FUNCTION_BLOCK FB_EventIoTExporter IMPLEMENTS InterfaceEventViewer
VAR_INPUT
	tzinfo : ST_TimeZoneInformation;
END_VAR
VAR_OUTPUT
	export_event : ST_EventView;
END_VAR
VAR
END_VAR

{warning 'add method implementation '}
METHOD clear : BOOL
END_METHOD

{warning 'add method implementation '}
METHOD history_clear : BOOL
END_METHOD

{warning 'add method implementation '}
METHOD send_event : BOOL
VAR_INPUT
	event_container	: REFERENCE TO EventContainer;
END_VAR
VAR
	iso_datetime : STRING;
	source_name : STRING;
END_VAR
IF event_container.event.bRaised THEN
	UTF8_TO_WSTRING(
		ADR(export_event.Computer),
		ADR(event_container.event.module_name),
		SIZEOF(export_event.Computer)
	);
	
	source_name := event_container.event.ipSourceInfo.sName;
	
	UTF8_TO_WSTRING(
		ADR(export_event.sSource),
		ADR(source_name),
		SIZEOF(export_event.sSource)
	);
	
	export_event.bConfirmable := event_container.event.eConfirmationState <> TcEventConfirmationState.NotSupported;
	CASE event_container.event.eSeverity OF 
		TcEventSeverity.Critical:
			export_event.Severity := "危険";		
		TcEventSeverity.Error:
			export_event.Severity := "異常";
		TcEventSeverity.Info:
			export_event.Severity := "情報";
		TcEventSeverity.Verbose:
			export_event.Severity := "ログ";
		TcEventSeverity.Warning:
			export_event.Severity := "警告";
		ELSE
			export_event.Severity := TO_WSTRING(event_container.event.eSeverity);
	END_CASE
	
	IF event_container.event.bRaised THEN 
		export_event.ConfirmState := "発生";
	ELSE
		export_event.ConfirmState := "解除";
	END_IF
	
	export_event.nEventId := event_container.event.nEventId;
	UTF8_TO_WSTRING(
		ADR(export_event.MessageText),
		ADR(event_container.event_text),
		SIZEOF(export_event.MessageText)
	);
	
	
	IF event_container.event.bRaised THEN
		iso_datetime := FILETIME64_TO_ISO8601(
							fileTime := event_container.event.nTimeRaised,
							nBias := TO_INT(tzInfo.bias), 
							bUTC :=TRUE, 
							nPrecision := 0
						);
	ELSE
		iso_datetime := FILETIME64_TO_ISO8601(
							fileTime := event_container.event.nTimeCleared,
							nBias := TO_INT(tzInfo.bias), 
							bUTC :=TRUE, 
							nPrecision := 0
						);	
	END_IF
	
	export_event.sDate := MID(iso_datetime, 10, 1);
	export_event.sTime := MID(iso_datetime, 8, 12);
END_IF
END_METHOD

{warning 'add method implementation '}
METHOD show : BOOL
VAR_INPUT
	event_container	: REFERENCE TO EventContainer;
END_VAR
END_METHOD

END_FUNCTION_BLOCK

(* stored: Version 1.1.0.1, ProductVersion 3.1.4024.15
   POU FB_EventIoTExporter: Id {8194870f-80e5-48cc-9062-7a48f44737ce}, SpecialFunc None
   Method clear: Id {e300ba77-2c0e-4b57-b938-50d10b136472}
   Method history_clear: Id {387e2cd7-0b47-433f-89e4-60da0f7a4953}
   Method send_event: Id {3b874412-bd46-4068-904a-e07474905b56}
   Method show: Id {85c5b3f3-7b74-4fc5-af14-9395b7991d3b} *)
